{attribute 'linkalways'} 
{attribute 'no_explicit_call' := 'This FB is a CLASS and must be accessed using methods or properties'}
{attribute 'enable_dynamic_creation'}
FUNCTION_BLOCK Node_ContainerType_Vector_TcVnVector3_REAL EXTENDS Node
VAR
    out : _GUID;
END_VAR

METHOD PUBLIC  Clone : I_Node
VAR
	pNode : POINTER TO Node_ContainerType_Vector_TcVnVector3_REAL;
END_VAR
pNode := __NEW(Node_ContainerType_Vector_TcVnVector3_REAL);
Clone := pNode^;
END_METHOD

METHOD FB_init : BOOL
VAR_INPUT
	bInitRetains : BOOL; // if TRUE, the retain variables are initialized (warm start / cold start)
	bInCopyCode : BOOL;  // if TRUE, the instance afterwards gets moved into the copy code (online change)
END_VAR
AddOutput('out', out);
END_METHOD

METHOD PROTECTED OnExecute
out.Value := ContainerType_Vector_TcVnVector3_REAL;
END_METHOD

END_FUNCTION_BLOCK

(* stored: Version 1.1.0.1, ProductVersion 3.1.4026.17
   POU Node_ContainerType_Vector_TcVnVector3_REAL: Id {56edc7cf-f196-08aa-0291-d84ed2348150}, SpecialFunc None
   Folder Constructor: Id {df508368-b644-0761-0c5e-a3d0c347e72d}
   Method Clone: Id {9fc58398-0688-08fa-2285-8842c3fcdfa2}
   Method FB_init: Id {7f9caba3-fbee-0096-38ab-0a9f1081e43c}
   Method OnExecute: Id {04d90a01-210b-068a-0a4a-3537077e60f4} *)
